// TwinCAT 3 PLC project Untitled1
// ProgramVersion: 3.1.4024.0
// libraries:
//   Tc2_MC2, * (Beckhoff Automation GmbH)
//   Tc2_Standard, * (Beckhoff Automation GmbH)
//   Tc2_System, * (Beckhoff Automation GmbH)
//   Tc3_Module, * (Beckhoff Automation GmbH)
// project tree:
//   GVLs/ GVL.TcGVL
//   / PlcTask.TcTTO
//   POUs/ MAIN.TcPOU
// real-time tasks:
//   TASK PlcTask: cycle T#10ms, priority 20, ADS port 350
// motion (NC):
//   TASK NC-Task 1 SAF: cycle T#2ms, priority 4, ADS port 501
//   TASK NC-Task 1 SVB: cycle T#10ms, priority 8, ADS port 511
//   AXIS Axis 1 (id 3)
//     OtherSettings: AllowMotionCmdToSlave=true
//     encoder EncType=1
//     drive DrvType=5
//       Analog: TorqueSetpointScale=10, ScaleFactorActTorque=0.1
//       TimeComp: TaskDelayCycles=1
//     controller CtrType=1
//       CtrPara: PriorControlFactor=1
//         Observer: BandWidth=20
//   AXIS Axis 2 (id 4)
//     OtherSettings: AllowMotionCmdToSlave=true
//     encoder EncType=1
//     drive DrvType=5
//       Analog: TorqueSetpointScale=10, ScaleFactorActTorque=0.1
//       TimeComp: TaskDelayCycles=1
//     controller CtrType=1
//       CtrPara: PriorControlFactor=1
//         Observer: BandWidth=20
// variable links:
//   Untitled1/Untitled1 Instance <-> NC-Task 1 SAF/Axes/Axis 1
//     PlcTask Inputs/GVL.Axis1.NcToPlc <-> Outputs/ToPlc
//     PlcTask Outputs/GVL.Axis1.PlcToNc <-> Inputs/FromPlc
//   Untitled1/Untitled1 Instance <-> NC-Task 1 SAF/Axes/Axis 2
//     PlcTask Inputs/GVL.Axis2.NcToPlc <-> Outputs/ToPlc
//     PlcTask Outputs/GVL.Axis2.PlcToNc <-> Inputs/FromPlc

CONFIGURATION Untitled1
    RESOURCE PLC ON TwinCAT3
        TASK PlcTask(INTERVAL := T#10ms, PRIORITY := 20);
        PROGRAM MAIN WITH PlcTask : MAIN;
    END_RESOURCE
END_CONFIGURATION

// ---- GVLs/GVL.TcGVL
{attribute 'qualified_only'}
VAR_GLOBAL
	Axis1 : AXIS_REF;
	Axis2 : AXIS_REF;
END_VAR

// ---- POUs/MAIN.TcPOU
PROGRAM MAIN
VAR
	Enable_Axis1: BOOL;
	Enable_Axis2: BOOL;
	Move_Axis1 : BOOL;
	Move_Axis2 : BOOL;
	Abilita_Axis1 : MC_Power;
	Abilita_Axis2 : MC_Power;
	Muovi_Axis1 : MC_MoveRelative;
	Muovi_Axis2 : MC_MoveRelative;
END_VAR

Abilita_Assi();
Muovi_Assi();

ACTION Abilita_Assi:
Abilita_Axis1(
	Axis:= GVL.Axis1, 
	Enable:= Enable_Axis1, 
	Enable_Positive:= TRUE, 
	Enable_Negative:= TRUE, 
	Override:= 100);

Abilita_Axis2(
	Axis:= GVL.Axis2, 
	Enable:= Enable_Axis2, 
	Enable_Positive:= TRUE, 
	Enable_Negative:= TRUE, 
	Override:= 100);
END_ACTION

ACTION Muovi_Assi:
Muovi_Axis1(
	Axis:= GVL.Axis1, 
	Execute:= Move_Axis1, 
	Distance:= 3600, 
	Velocity:= 9000 );
	
Muovi_Axis1(
	Axis:= GVL.Axis2, 
	Execute:= Move_Axis2, 
	Distance:= 3600, 
	Velocity:= 9000 );
END_ACTION

END_PROGRAM
